// TwinCAT 3 PLC project PalletLift12
// ProgramVersion: 3.1.4026.10
// CompilerDefines: VISU_USEPROPERTYINFO
// libraries:
//   Tc2_Standard, * (Beckhoff Automation GmbH)
//   Tc2_System, * (Beckhoff Automation GmbH)
// project tree:
//   / GlobalTextList.TcGTLO, PlcTask.TcTTO, Visualization Manager.TcVMO (not stored)
//   GVLs/ GVL.TcGVL
//   POUs/ MAIN.TcPOU, MotorCylinder.TcPOU, Sensor.TcPOU, Simulation.TcPOU, Switch.TcPOU
//   VISUs/ Visualization.TcVIS
// real-time tasks:
//   TASK PlcTask: cycle T#10ms, priority 20, ADS port 350

CONFIGURATION PalletLift12
    RESOURCE PLC ON TwinCAT3
        TASK PlcTask(INTERVAL := T#10ms, PRIORITY := 20);
        PROGRAM MAIN WITH PlcTask : MAIN;
        PROGRAM Simulation WITH PlcTask : Simulation;
    END_RESOURCE
END_CONFIGURATION

// ---- GVLs/GVL.TcGVL
{attribute 'qualified_only'}
VAR_GLOBAL
	_ExtendButton			:Switch();
	_RetractButton			:Switch();
	_Cylinder				:MotorCylinder(CylinderMaxLength := 500.0);
	_UpLimitSensor			:Sensor();
	_DownLimitSensor		:Sensor();
END_VAR

// ---- POUs/MAIN.TcPOU
PROGRAM MAIN
VAR
END_VAR

IF GVL._ExtendButton.IsPressed AND NOT GVL._UpLimitSensor.Triggered THEN
	GVL._Cylinder.RotateMotorExtend := TRUE;
ELSIF GVL._ExtendButton.IsPressed AND GVL._UpLimitSensor.Triggered THEN
	{warning 'Table reached the upper limit, can not lift further'}
	//Tähän joku koodi että sama teksti ei tulostu joka syklillä jos nappula pidetään pohjassa
END_IF

IF GVL._RetractButton.IsPressed AND NOT GVL._DownLimitSensor.Triggered THEN
	GVL._Cylinder.Retract := TRUE;
ELSIF GVL._RetractButton.IsPressed AND GVL._DownLimitSensor.Triggered THEN
	{warning 'Table reached the lower limit, can not depress further'}
	//Tähän joku koodi että sama teksti ei tulostu joka syklillä jos nappula pidetään pohjassa
END_IF

END_PROGRAM

// ---- POUs/Simulation.TcPOU
PROGRAM Simulation
VAR
	_CylinderDistance		:REAL;
END_VAR

GVL._Cylinder.CylinderDistance := _CylinderDistance;

IF GVL._Cylinder.Extend THEN
	_CylinderDistance := _CylinderDistance + 0.1;
ELSIF GVL._Cylinder.Retract THEN
	_CylinderDistance := _CylinderDistance - 0.1;
END_IF

END_PROGRAM

// ---- POUs/Switch.TcPOU
FUNCTION_BLOCK Switch
VAR_INPUT
END_VAR
VAR_OUTPUT
END_VAR
VAR
END_VAR

METHOD PUBLIC IsPressed : BOOL
VAR_INPUT
END_VAR
END_METHOD

END_FUNCTION_BLOCK

// ---- POUs/MotorCylinder.TcPOU
FUNCTION_BLOCK MotorCylinder
VAR
END_VAR
VAR_INPUT
	_CylinderMaxLength		:REAL; //In mm
END_VAR

//Cylinder distance in mm, as if measured by the motor cylinder assembly

PROPERTY PUBLIC CylinderDistance : REAL
GET
END_GET
SET
END_SET
END_PROPERTY

// Returns true if extending is possible
METHOD PUBLIC Extend : BOOL
VAR_INPUT
END_VAR
IF NOT IsFullyExtended() THEN
	RotateMotorExtend := TRUE;
	Extend := TRUE;
ELSE
	Extend := FALSE;
END_IF
END_METHOD

METHOD PRIVATE IsFullyExtended : BOOL
IF _CylinderDistance >= 100 THEN
	IsFullyExtended := TRUE;
END_IF
END_METHOD

METHOD PRIVATE IsFullyRetracted : BOOL
IF _CylinderDistance <= 0 THEN
	IsFullyRetracted := TRUE;
END_IF
END_METHOD

METHOD PUBLIC Retract : BOOL
VAR_INPUT
END_VAR
END_METHOD

PROPERTY PUBLIC RotateMotorExtend : BOOL
SET
END_SET
END_PROPERTY

END_FUNCTION_BLOCK

// ---- POUs/Sensor.TcPOU
FUNCTION_BLOCK Sensor
VAR
END_VAR

PROPERTY PUBLIC Triggered : BOOL
GET
END_GET
END_PROPERTY

END_FUNCTION_BLOCK

// ---- VISUs/Visualization.TcVIS
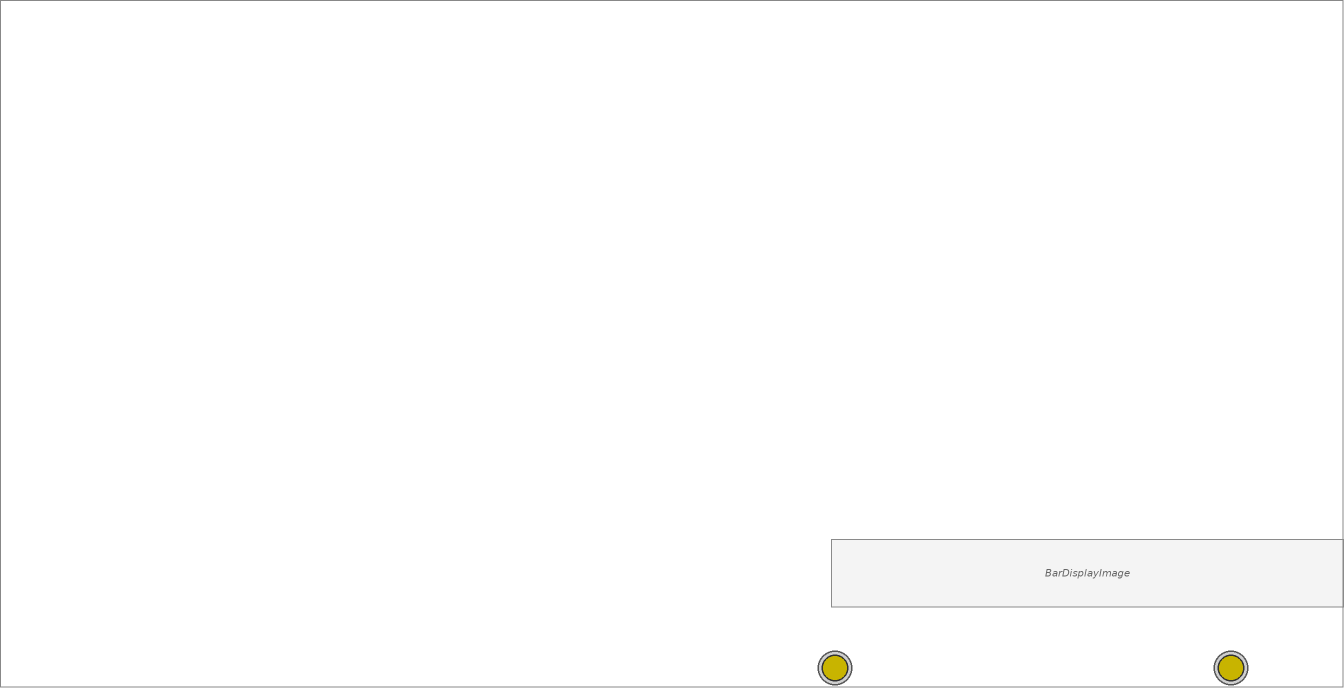
VISUALIZATION Visualization  // 1344x688
    BarDisplayImage (831,539 513x68), style: BarDisplayImage-Gray, scale format: %.1f, scale 0..100
    Lamp1 (815,648 40x40), style: Lamp-Lamp1-Yellow
    Lamp1 (1211,648 40x40), style: Lamp-Lamp1-Yellow
END_VISUALIZATION
